// TIA Portal V17 export
// export: Created 2023-04-04T07:45:38.0406474Z, ExportSetting WithDefaults, DisplayName Totally Integrated Automation Portal, DisplayVersion V17 Update 4, DisplayName TIA Portal Openness, DisplayVersion V17 Update 4, DisplayName TIA Portal Version Control Interface, DisplayVersion V17, DisplayName STEP 7 Professional, DisplayVersion V17 Update 4, DisplayName STEP 7 Safety, DisplayVersion V17, DisplayName WinCC Professional, DisplayVersion V17 Update 4
DATA_BLOCK "SM_TEST"   // DB9
{ S7_Optimized_Access := 'TRUE' }
VERSION : 0.1
// stored: AutoNumber true, DBAccessibleFromOPCUA true, DBAccessibleFromWebserver true, IsOnlyStoredInLoadMemory false, IsRetainMemResEnabled false, IsWriteProtectedInAS false, MemoryReserve 100
   VAR
      xEnable_comm : Bool;
      xComm_enabled : Bool;
      xSS1_fault : Bool;
      xAutoCharge_command : Bool;
      xSM1_readyCondition : Bool;
      xSystem_ready : Bool;
      "xBattery_cl/op_command" : Bool;
      xBypass_Estop : Bool;
   END_VAR
BEGIN
END_DATA_BLOCK
